PROGRAM P2_04_Cleaning_Ctrl
VAR
	bPreCleaning_Active				:BOOL;
	bMainCleaning_Active			:BOOL;
	bRinsing_Active					:BOOL;
	bPWCleaning_Active				:BOOL;
	bDraining_Active				:BOOL;
	bBlowing_Active					:BOOL;
	bControl_Active					:BOOL;
END_VAR

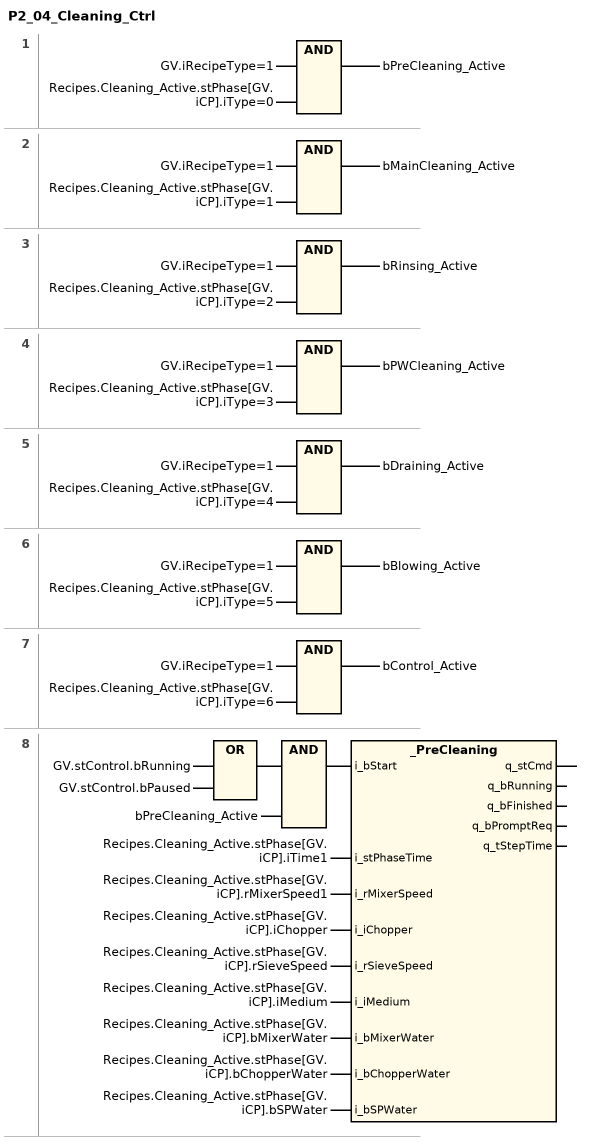
// NETWORK 1
bPreCleaning_Active := (GV.iRecipeType=1) AND (Recipes.Cleaning_Active.stPhase[GV.iCP].iType=0);

// NETWORK 2
bMainCleaning_Active := (GV.iRecipeType=1) AND (Recipes.Cleaning_Active.stPhase[GV.iCP].iType=1);

// NETWORK 3
bRinsing_Active := (GV.iRecipeType=1) AND (Recipes.Cleaning_Active.stPhase[GV.iCP].iType=2);

// NETWORK 4
bPWCleaning_Active := (GV.iRecipeType=1) AND (Recipes.Cleaning_Active.stPhase[GV.iCP].iType=3);

// NETWORK 5
bDraining_Active := (GV.iRecipeType=1) AND (Recipes.Cleaning_Active.stPhase[GV.iCP].iType=4);

// NETWORK 6
bBlowing_Active := (GV.iRecipeType=1) AND (Recipes.Cleaning_Active.stPhase[GV.iCP].iType=5);

// NETWORK 7
bControl_Active := (GV.iRecipeType=1) AND (Recipes.Cleaning_Active.stPhase[GV.iCP].iType=6);

// NETWORK 8
_PreCleaning(i_bStart := (GV.stControl.bRunning OR GV.stControl.bPaused) AND bPreCleaning_Active, i_stPhaseTime := Recipes.Cleaning_Active.stPhase[GV.iCP].iTime1, i_rMixerSpeed := Recipes.Cleaning_Active.stPhase[GV.iCP].rMixerSpeed1, i_iChopper := Recipes.Cleaning_Active.stPhase[GV.iCP].iChopper, i_rSieveSpeed := Recipes.Cleaning_Active.stPhase[GV.iCP].rSieveSpeed, i_iMedium := Recipes.Cleaning_Active.stPhase[GV.iCP].iMedium, i_bMixerWater := Recipes.Cleaning_Active.stPhase[GV.iCP].bMixerWater, i_bChopperWater := Recipes.Cleaning_Active.stPhase[GV.iCP].bChopperWater, i_bSPWater := Recipes.Cleaning_Active.stPhase[GV.iCP].bSPWater);

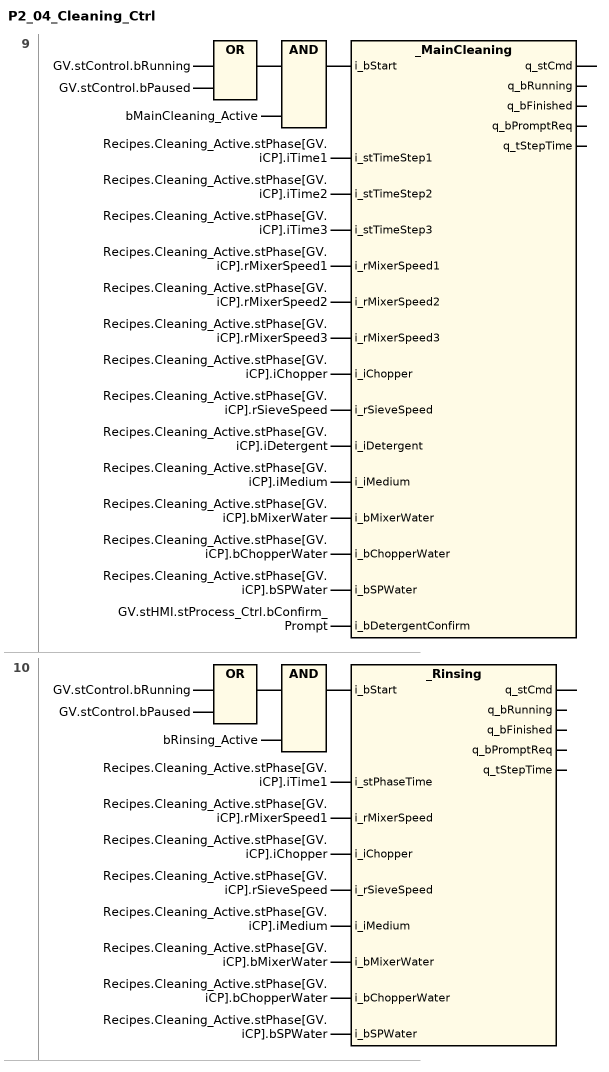
// NETWORK 9
_MainCleaning(i_bStart := (GV.stControl.bRunning OR GV.stControl.bPaused) AND bMainCleaning_Active, i_stTimeStep1 := Recipes.Cleaning_Active.stPhase[GV.iCP].iTime1, i_stTimeStep2 := Recipes.Cleaning_Active.stPhase[GV.iCP].iTime2, i_stTimeStep3 := Recipes.Cleaning_Active.stPhase[GV.iCP].iTime3, i_rMixerSpeed1 := Recipes.Cleaning_Active.stPhase[GV.iCP].rMixerSpeed1, i_rMixerSpeed2 := Recipes.Cleaning_Active.stPhase[GV.iCP].rMixerSpeed2, i_rMixerSpeed3 := Recipes.Cleaning_Active.stPhase[GV.iCP].rMixerSpeed3, i_iChopper := Recipes.Cleaning_Active.stPhase[GV.iCP].iChopper, i_rSieveSpeed := Recipes.Cleaning_Active.stPhase[GV.iCP].rSieveSpeed, i_iDetergent := Recipes.Cleaning_Active.stPhase[GV.iCP].iDetergent, i_iMedium := Recipes.Cleaning_Active.stPhase[GV.iCP].iMedium, i_bMixerWater := Recipes.Cleaning_Active.stPhase[GV.iCP].bMixerWater, i_bChopperWater := Recipes.Cleaning_Active.stPhase[GV.iCP].bChopperWater, i_bSPWater := Recipes.Cleaning_Active.stPhase[GV.iCP].bSPWater, i_bDetergentConfirm := GV.stHMI.stProcess_Ctrl.bConfirm_Prompt);

// NETWORK 10
_Rinsing(i_bStart := (GV.stControl.bRunning OR GV.stControl.bPaused) AND bRinsing_Active, i_stPhaseTime := Recipes.Cleaning_Active.stPhase[GV.iCP].iTime1, i_rMixerSpeed := Recipes.Cleaning_Active.stPhase[GV.iCP].rMixerSpeed1, i_iChopper := Recipes.Cleaning_Active.stPhase[GV.iCP].iChopper, i_rSieveSpeed := Recipes.Cleaning_Active.stPhase[GV.iCP].rSieveSpeed, i_iMedium := Recipes.Cleaning_Active.stPhase[GV.iCP].iMedium, i_bMixerWater := Recipes.Cleaning_Active.stPhase[GV.iCP].bMixerWater, i_bChopperWater := Recipes.Cleaning_Active.stPhase[GV.iCP].bChopperWater, i_bSPWater := Recipes.Cleaning_Active.stPhase[GV.iCP].bSPWater);

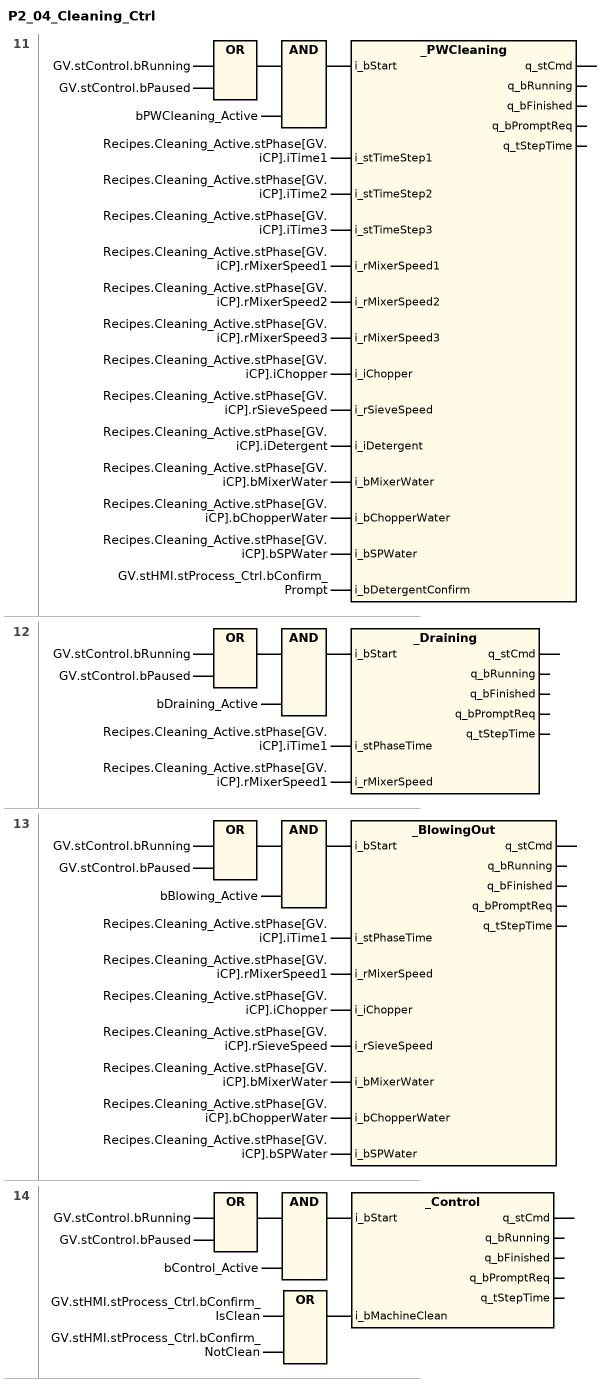
// NETWORK 11
_PWCleaning(i_bStart := (GV.stControl.bRunning OR GV.stControl.bPaused) AND bPWCleaning_Active, i_stTimeStep1 := Recipes.Cleaning_Active.stPhase[GV.iCP].iTime1, i_stTimeStep2 := Recipes.Cleaning_Active.stPhase[GV.iCP].iTime2, i_stTimeStep3 := Recipes.Cleaning_Active.stPhase[GV.iCP].iTime3, i_rMixerSpeed1 := Recipes.Cleaning_Active.stPhase[GV.iCP].rMixerSpeed1, i_rMixerSpeed2 := Recipes.Cleaning_Active.stPhase[GV.iCP].rMixerSpeed2, i_rMixerSpeed3 := Recipes.Cleaning_Active.stPhase[GV.iCP].rMixerSpeed3, i_iChopper := Recipes.Cleaning_Active.stPhase[GV.iCP].iChopper, i_rSieveSpeed := Recipes.Cleaning_Active.stPhase[GV.iCP].rSieveSpeed, i_iDetergent := Recipes.Cleaning_Active.stPhase[GV.iCP].iDetergent, i_bMixerWater := Recipes.Cleaning_Active.stPhase[GV.iCP].bMixerWater, i_bChopperWater := Recipes.Cleaning_Active.stPhase[GV.iCP].bChopperWater, i_bSPWater := Recipes.Cleaning_Active.stPhase[GV.iCP].bSPWater, i_bDetergentConfirm := GV.stHMI.stProcess_Ctrl.bConfirm_Prompt);

// NETWORK 12
_Draining(i_bStart := (GV.stControl.bRunning OR GV.stControl.bPaused) AND bDraining_Active, i_stPhaseTime := Recipes.Cleaning_Active.stPhase[GV.iCP].iTime1, i_rMixerSpeed := Recipes.Cleaning_Active.stPhase[GV.iCP].rMixerSpeed1);

// NETWORK 13
_BlowingOut(i_bStart := (GV.stControl.bRunning OR GV.stControl.bPaused) AND bBlowing_Active, i_stPhaseTime := Recipes.Cleaning_Active.stPhase[GV.iCP].iTime1, i_rMixerSpeed := Recipes.Cleaning_Active.stPhase[GV.iCP].rMixerSpeed1, i_iChopper := Recipes.Cleaning_Active.stPhase[GV.iCP].iChopper, i_rSieveSpeed := Recipes.Cleaning_Active.stPhase[GV.iCP].rSieveSpeed, i_bMixerWater := Recipes.Cleaning_Active.stPhase[GV.iCP].bMixerWater, i_bChopperWater := Recipes.Cleaning_Active.stPhase[GV.iCP].bChopperWater, i_bSPWater := Recipes.Cleaning_Active.stPhase[GV.iCP].bSPWater);

// NETWORK 14
_Control(i_bStart := (GV.stControl.bRunning OR GV.stControl.bPaused) AND bControl_Active, i_bMachineClean := GV.stHMI.stProcess_Ctrl.bConfirm_IsClean OR GV.stHMI.stProcess_Ctrl.bConfirm_NotClean);

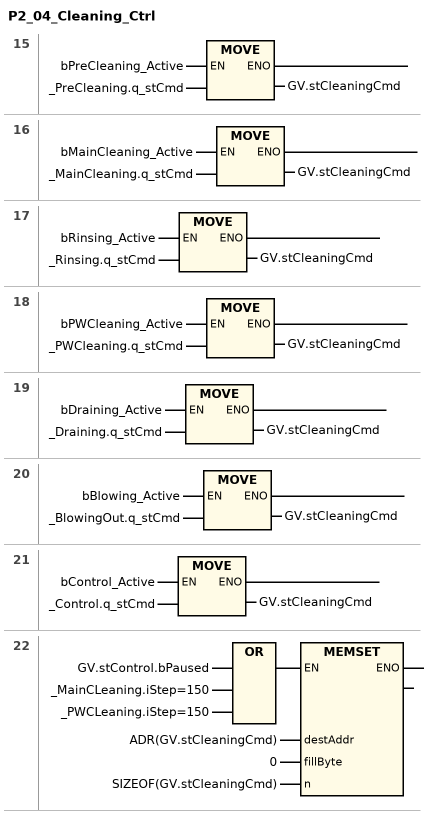
// NETWORK 15
IF bPreCleaning_Active THEN GV.stCleaningCmd := _PreCleaning.q_stCmd; END_IF

// NETWORK 16
IF bMainCleaning_Active THEN GV.stCleaningCmd := _MainCleaning.q_stCmd; END_IF

// NETWORK 17
IF bRinsing_Active THEN GV.stCleaningCmd := _Rinsing.q_stCmd; END_IF

// NETWORK 18
IF bPWCleaning_Active THEN GV.stCleaningCmd := _PWCleaning.q_stCmd; END_IF

// NETWORK 19
IF bDraining_Active THEN GV.stCleaningCmd := _Draining.q_stCmd; END_IF

// NETWORK 20
IF bBlowing_Active THEN GV.stCleaningCmd := _BlowingOut.q_stCmd; END_IF

// NETWORK 21
IF bControl_Active THEN GV.stCleaningCmd := _Control.q_stCmd; END_IF

// NETWORK 22
IF GV.stControl.bPaused OR (_MainCLeaning.iStep=150) OR (_PWCLeaning.iStep=150) THEN
    MEMSET(destAddr := ADR(GV.stCleaningCmd), fillByte := 0, n := SIZEOF(GV.stCleaningCmd));
END_IF

END_PROGRAM

(* stored: Version 1.1.0.1, ProductVersion 3.1.4026.13
   POU P2_04_Cleaning_Ctrl: Id {626edb41-8728-41d4-a27c-0fd2a6981518}, SpecialFunc None *)
